PROGRAM SafetyCheck
VAR
	// slave robot information, including arm status and cartesian data
	m_slaveStatus AT %I* :ST_slaveStatus;
	
	// slave robot joint data
	m_slaveJointData AT %I* :ST_slaveJointData;
	
	// setup robot information
	m_setupStatus AT %I* :ST_SetupStatus;
	
	// setup robot joint data
	m_setupJointsData AT %I* :ST_SetupJointData;
	
	// error check result
	m_safetyCheckData AT %Q* :ST_SafetyData;
	
	m_initFlag:bool;
	m_cartCheck :FB_CartCheck;
	m_setupArmCheck:FB_SetupArmCheck;
	m_slaveArmCheck:FB_SlaveArmCheck;
	
	i: INT;
END_VAR

// reset data
IF FALSE = m_initFlag  THEN
	FOR i:=1  TO g_sArmNum DO 
		m_safetyCheckData.m_slaveErrFlag[i]:=FALSE;
		m_safetyCheckData.m_setupErrFlag[i]:=FALSE;
		m_safetyCheckData.m_cartErrFlag:=false;
	END_FOR
	m_initFlag:=TRUE;
END_IF

m_slaveArmCheck.check(m_slaveStatus,m_slaveJointData, o_errorFlag=>m_safetyCheckData.m_slaveErrFlag);
m_setupArmCheck.check(m_setupStatus,m_setupJointsData, o_errorFlag=>m_safetyCheckData.m_setupErrFlag);

END_PROGRAM

(* stored: Version 1.1.0.1, ProductVersion 3.1.4024.11
   POU SafetyCheck: Id {54e6e883-3f22-4a40-9066-2b433bf8009c}, SpecialFunc None *)
